(* IEC 61131-3 sources: demo-MpCnc-with-mapp-motion/Motion/Cnc, 4 files *)

(* ---- Cyclic.st ---- *)
PROGRAM _CYCLIC
	MpCnc3Axis_0();

	g_positionX := MpCnc3Axis_0.X;
	g_positionY := MpCnc3Axis_0.Y;

	IF MFunc_CutterUp THEN
		MFunc_CutterUp := FALSE;
	END_IF

	IF MFunc_CutterDown THEN
		MFunc_CutterDown := FALSE;
	END_IF
END_PROGRAM

(* ---- Exit.st ---- *)
PROGRAM _EXIT
	MpCnc3Axis_0.Enable := FALSE;
    MpCnc3Axis_0.Power  := FALSE;
    MpCnc3Axis_0.Home   := FALSE;
    MpCnc3Axis_0();

END_PROGRAM

(* ---- Init.st ---- *)
PROGRAM _INIT
	MpCnc3Axis_0.MpLink := ADR(gCncXYZ);
	MpCnc3Axis_0.Enable := TRUE;
	MpCnc3Axis_0.Parameters := ADR(CncParameters);

	MpCnc3Axis_0.Override := 100.0;

	CncParameters.ProgramName := 'Micky';

END_PROGRAM

(* ---- Variables.var ---- *)
VAR
	MFunc_CutterDown : BOOL;
	MFunc_CutterUp : BOOL;
	MpCnc3Axis_0 : MpCnc3Axis;
	CncParameters : MpCnc2AxisParType;
END_VAR
